{attribute 'linkalways'} 
{attribute 'no_explicit_call' := 'This FB is a CLASS and must be accessed using methods or properties'}
{attribute 'enable_dynamic_creation'}
FUNCTION_BLOCK SynchronousRpcHandlers IMPLEMENTS I_SynchronousRpcHandlers
VAR
	handlers : Dictionary;
	_hasHandlers : BOOL;
END_VAR

PROPERTY PUBLIC HasHandlers : BOOL
GET
HasHandlers := _hasHandlers;
END_GET
END_PROPERTY

METHOD PUBLIC RegisterHandler
VAR_INPUT
	MethodName : T_MAXSTRING;
	Handler : I_SynchronousRpcHandler;
END_VAR
handlers.AddOrUpdate(MethodName, Handler);
_hasHandlers := true;
END_METHOD

METHOD PUBLIC TryGetByMethodName : BOOL
VAR_INPUT
	MethodName : T_MAXSTRING;
	Destination : REFERENCE TO I_SynchronousRpcHandler;
END_VAR
TryGetByMethodName := handlers.TryGetValue(MethodName, Destination);
END_METHOD

END_FUNCTION_BLOCK

(* stored: Version 1.1.0.1, ProductVersion 3.1.4024.12
   POU SynchronousRpcHandlers: Id {cdfb1c94-3217-037e-37e9-3e856bc4db90}, SpecialFunc None
   Property HasHandlers: Id {2605a19b-dc3f-44fb-9955-a556daab8d19}
   Get Get: Id {19d45a51-bd11-4b50-8fa5-b20303b75f89}
   Method RegisterHandler: Id {609e53c5-acdf-01aa-0656-3cf6fac1acc2}
   Method TryGetByMethodName: Id {9f3d7a27-ca03-0efa-0266-b6d155dc3dde} *)
